INTERFACE I_PersistentEventStorage

METHOD StoreEvent
VAR_INPUT
	stEvent : ST_Event;
END_VAR
END_METHOD

END_INTERFACE

(* stored: Version 1.1.0.1, ProductVersion 3.1.4024.12
   Itf I_PersistentEventStorage: Id {6266317a-6090-4b13-87bf-5be655b4132b}
   Method StoreEvent: Id {845ca985-27f9-4541-99e5-49c045548917} *)
